# B&R Automation Studio project Cognex_V1_5
Automation Studio 4.6.3.55 SP

## Configuration PP500_15

CPU , AutomationRuntime H4.06, Build 4.1.2, Safety 1.6, Vc V4.05.6

### Task classes (Cpu.sw)
```
Cyclic#8:
  Cognex <- Cognex.prg
  CognexVisN <- CognexVisNativeMode.prg
  CognexVisC <- CognexVisCommissioning.prg
  CognexVisA <- CognexVisArchive.prg
  CognexVisM <- CognexVisMain.prg
VcDataObjects: Visu <- Visu.dob
Binaries: vcclbox, vcctext, vcrt, vcresman, vccbar, vccstr, vccurl, vcchtml, vcpfmtcx, vcptelo, vcfile, vcdsint, vcpdsw, vccshape, arial, vccbmp, vcmgr, vcpdi855, vcshared, Visu01, vcdsloc, vcfntttf, vccovl, vctcal, arialbd, vcalarm, vcpfpp50, vccnum, vccline, vcpdi815, vccbtn, vcgclass, vcbclass, vcxml, Visu02, Visu03, visvc, vcpdvnc, vcnet, arconfig, sysconf, ashwd, asfw, iomap, vccalarm
Libraries: asieccon, asstring, astime, runtime, FileIO, Visapi, standard, BR_ATL_BMP, BR_ATL_LOG, sys_lib, dataobj, BR_ATL_COG, AsTCP, ethernet, AsICMP
```

## Configuration X20CPU1484

CPU , AutomationRuntime V3.08, Build 4.1.2, Vc V3.95.6

### Task classes (Cpu.sw)
```
Cyclic#8 (cycle 4000 us, tolerance 30004000 us):
  Cognex <- Cognex.prg
  CognexVisM <- CognexVisMain.prg
  CognexVisA <- CognexVisArchive.prg
  CognexVisN <- CognexVisNativeMode.prg
VcDataObjects: Visu <- Visu.dob
Binaries: vcdsint, vcclbox, Visu03, vcctext, vcrt, vccnum, vccbar, vccstr, vccurl, vcchtml, vcresman, vcfile, vcpfx20, vcpdsw, vccshape, arial, vccbmp, vcmgr, visvc, Visu01, vcdsloc, vcfntttf, vccovl, vctcal, arialbd, vcalarm, vccline, vcshared, vccbtn, vcgclass, vcbclass, vcxml, vcnet, vcpdvnc, Visu02, ashwd, sysconf, asfw, arconfig, iomap
Libraries: sys_lib, asstring, BR_ATL_LOG, Operator, Runtime, AsTime, AsIecCon, FileIO, Visapi, standard, BR_ATL_BMP, ashw, dataobj, BR_ATL_COG, AsTCP
```

### Hardware
```
In-Sight : FBE.0000031D_In-Sight-7000 v1.0 (OrderNumber=In-Sight)  [PLK1 -> PLC1.IF3 (NodeNumber=1)]
  Supervision = off
  p2000s01_direction = wo
  p2000s02_direction = wo
  p2001s01_direction = ro
  p2001s02_direction = ro
  p2010s01_direction = ro
  p2011s01_direction = ro
  p2011s02_direction = ro
  p2011s03_direction = ro
  p2011s04_direction = ro
  p2011s05_direction = ro
  p2011s06_direction = ro
  p2011s07_direction = ro
  p2011s08_direction = ro
  p2011s09_direction = ro
  p2011s0A_direction = ro
  p2011s0B_direction = ro
  p2021s01_direction = wo
  p2021s02_direction = wo
  p2021s03_direction = wo
  p2030s01_value = 1500
PLC1 : X20CP1486 v1.1.2.0
  Connector IF2:
    ActivateDevice = 1
    Mode = DHCP Server
    InternetAddress = 192.168.0.10
    SubnetMask = 255.255.255.0
    Lease1
    LeaseName1 = Cognex
    LeaseStartAddress1 = 192.168.0.50
    LeaseStopAddress1 = 192.168.0.55
    LeaseSubnetMask1 = 255.255.255.0
    Vnc1
    VncVcObjectName1 = Visu
    VncPortNumber1 = 5900
    VncMaxConnections1 = 1
    VncRefreshRate1 = 500
    VncConnectionTimeout1 = 4
    VncAuthentication1 = 1
    VncPasswordViewOnly1 = r
    VncPasswordViewControl1 = w
  Connector IF3:
    MtuSize = 1500
    CycleTime = 800
    InternetAddress = 192.168.2.1
    SubnetMask = 255.255.255.0
  UserRamSize = 100000
  RemMemSize = 32000
  Connections = 6
  TimerDeviceType = EPLX2X
  TaskClassIdleTime = 800
  Cyclic1Duration = 2400
  Cyclic1Tolerance = 12000
  Cyclic3Duration = 50400
  Cyclic3Tolerance = 50400
  Cyclic8Duration = 4000
  Cyclic8Tolerance = 30004000
  TimerDevice = PLC1.IF3
```

### IoMap.iom - PLC1/IoMap.iom
```iecst
(********************************************************************
 * COPYRIGHT --
 ********************************************************************
 * File: IoMap.iom
 * Author: strickers
 * Created: May 07, 2012
 ********************************************************************
 * IO mapping file
 ********************************************************************)
VAR_CONFIG
	CognexVisM:CameraIsConnected AT %IX."In-Sight".ModuleOk;
	Cognex:tmpBarcodeRead1 AT %ID."In-Sight".InspectionResults_I2011_S01;
	Cognex:tmpBarcodeRead2 AT %ID."In-Sight".InspectionResults_I2011_S02;
	Cognex:tmpBarcodeRead3 AT %ID."In-Sight".InspectionResults_I2011_S03;
	Cognex:tmpBarcodeWrite1 AT %QD."In-Sight".UserData_I2021_S01;
	Cognex:tmpBarcodeWrite2 AT %QD."In-Sight".UserData_I2021_S02;
	Cognex:tmpBarcodeWrite3 AT %QD."In-Sight".UserData_I2021_S03;
	Cognex:cognex1cmd AT %QD."In-Sight".Control_I2000_S01;
	cognex_1.cmd.job_id AT %QW."In-Sight".JobLoadID_I2000_S02;
	Cognex:cognex1sta AT %ID."In-Sight".Status_I2001_S01;
	cognex_1.sta.job_id AT %IW."In-Sight".CurrentJobID_I2001_S02;
	Cognex:tmpTextRead1 AT %ID."In-Sight".InspectionResults_I2011_S04;
	Cognex:tmpTextRead2 AT %ID."In-Sight".InspectionResults_I2011_S05;
	Cognex:tmpTextRead3 AT %ID."In-Sight".InspectionResults_I2011_S06;
	Cognex:tmpData1 AT %ID."In-Sight".InspectionResults_I2011_S07;
	Cognex:tmpData2 AT %ID."In-Sight".InspectionResults_I2011_S08;
	Cognex:tmpData3 AT %ID."In-Sight".InspectionResults_I2011_S09;
	Cognex:tmpData4 AT %ID."In-Sight".InspectionResults_I2011_S0A;
	Cognex:tmpData5 AT %ID."In-Sight".InspectionResults_I2011_S0B;
END_VAR
```

## Logical view

Binary libraries used (declarations not repeated): AsICMP

### Global.typ
```iecst
(********************************************************************
 * COPYRIGHT --
 ********************************************************************
 * File: Global.typ
 * Author: strickers
 * Created: May 02, 2012
 ********************************************************************
 * Global data types of project Cognex_1
 ********************************************************************)

TYPE
	cognex_sta_typ : 	STRUCT
		connected_eth : BOOL;
		connected_plk : BOOL;
		trigger_ready : BOOL;
		trigger_ack : BOOL;
		acquiring : BOOL;
		missed_acq : BOOL;
		offline_reason : USINT;
		online : BOOL;
		inspecting : BOOL;
		inspecting_complete : BOOL;
		results_buffer_overrun : BOOL;
		results_valid : BOOL;
		job_loading : BOOL;
		job_load_complete : BOOL;
		job_load_failed : BOOL;
		set_user_data_ack : BOOL;
		exposure_complete : BOOL;
		soft_event_ack : USINT;
		job_id : UINT;
	END_STRUCT;
	cognex_cmd_typ : 	STRUCT
		trigger_enable : BOOL;
		trigger : BOOL;
		buffer_result_enable : BOOL;
		inspection_result_ack : BOOL;
		init_job_load : BOOL;
		set_offline : BOOL;
		set_user_data : BOOL;
		clr_exposure_complete : BOOL;
		soft_event : USINT;
		job_id : UINT;
		ping_camera : BOOL;
	END_STRUCT;
	cognex_typ : 	STRUCT
		cmd : cognex_cmd_typ;
		sta : cognex_sta_typ;
	END_STRUCT;
END_TYPE
```

### Global.var
```iecst
(*-------------------------------------------------------------------------------------------------------------------------------------------------------------------------------------------------------------------------*)
VAR
	cognex_1 : cognex_typ; (*Cognex main structure*)
	logbook : ARRAY[0..19] OF STRING[80];
END_VAR
(*-------------------------------------------------------------------------------------------------------------------------------------------------------------------------------------------------------------------------*)
VAR CONSTANT
	PictureWidth : UINT := 200; (*Cognex picture width*)
	PictureHeight : UINT := 150; (*Cognex picture height*)
END_VAR
VAR
	CognexPlkNode : STRING[3] := '1'; (*Powerlink node number for Cognex camera*)
	CognexEthIP : STRING[30] := '192.168.0.220'; (*IP address for camera when connected to Ethernet port*)
END_VAR
(*-------------------------------------------------------------------------------------------------------------------------------------------------------------------------------------------------------------------------*)
VAR
	VIS_HIDDEN : UINT := 1; (*Visualization status constants*)
END_VAR
VAR CONSTANT
	VIS_INACTIVE : UINT := 2;
	VIS_ACTIVE : UINT := 0;
END_VAR
(*-------------------------------------------------------------------------------------------------------------------------------------------------------------------------------------------------------------------------*)
VAR CONSTANT
	READ_ID1 : USINT := 1;
	READ_CFG : USINT := 2;
	WRITE_ID1 : USINT := 1;
	WRITE_ID2 : USINT := 2;
	WRITE_ID3 : USINT := 3;
	WRITE_CFG : USINT := 4;
END_VAR
(*-------------------------------------------------------------------------------------------------------------------------------------------------------------------------------------------------------------------------*)
VAR CONSTANT
	NONE : USINT := 0;
	CMD_INFO : USINT := 1;
	CMD_STATUS : USINT := 2;
	CMD_DELETE_JOBID3 : USINT := 3;
	CMD_SET_OFFLINE : USINT := 4;
END_VAR
```

### Program Logical/Cognex

#### Cognex.ab
```automation-basic
(********************************************************************
 * COPYRIGHT --
 ********************************************************************
 * Program: NewProgram
 * File: NewProgram.ab
 * Author: strickers
 * Version: 1.0
 * This task has the following purpose
 * - Transfer text string from sample into PLC variable
 * - Transfer barcode string from sample into PLC variable
 * - Transfer compare string to Cognex variable
 * - Transfer add on data (pass, angle, time) into PLC variables
 * - Transfer camera status into bool structure
 * - Transfer camera commands from PLC structure to camera
 ********************************************************************)

PROGRAM _INIT
		strcpy(ADR(strBarcodeWrite), ADR("ABA122"))
END_PROGRAM

PROGRAM _CYCLIC
	(* -------------------------------------------------------------------- *)
	(* Send ping to camera			 										*)
	IF (cognex_1.cmd.ping_camera) THEN
		ICMPping_0.enable 	= 1
		ICMPping_0.pHost 	= adr(CognexEthIP)
		ICMPping_0.timeout 	= 20
		ICMPping_0 FUB IcmpPing()
		IF(ICMPping_0.status <> 65535) THEN
			cognex_1.cmd.ping_camera = 0
			IF(ICMPping_0.status = 0) THEN
				cognex_1.sta.connected_eth = 1
			ELSE
				cognex_1.sta.connected_eth = 0
			ENDIF
		ENDIF
	ENDIF

	IF(cognex_1.sta.online) THEN
	(* -------------------------------------------------------------------- *)
	(* Transfer text string			 										*)
	memcpy(ADR(strTextRead)+0,ADR(tmpTextRead1), 4)
	memcpy(ADR(strTextRead)+4,ADR(tmpTextRead2), 4)
	memcpy(ADR(strTextRead)+8,ADR(tmpTextRead3), 4)

	(* -------------------------------------------------------------------- *)
	(* Transfer barcode string			 									*)
	memcpy(ADR(strBarcodeRead)+0,ADR(tmpBarcodeRead1), 4)
	memcpy(ADR(strBarcodeRead)+4,ADR(tmpBarcodeRead2), 4)
	memcpy(ADR(strBarcodeRead)+8,ADR(tmpBarcodeRead3), 4)

	memcpy(ADR(tmpBarcodeWrite1), ADR(strBarcodeWrite)+0, 4)
	memcpy(ADR(tmpBarcodeWrite2), ADR(strBarcodeWrite)+4, 4)
	memcpy(ADR(tmpBarcodeWrite3), ADR(strBarcodeWrite)+8, 4)
	IF(strcmp(ADR(strBarcodeWrite), ADR(strBarcodeWriteOld)) <> 0) THEN
		cognex_1.cmd.set_user_data = 1
		strcpy(ADR(strBarcodeWriteOld), ADR(strBarcodeWrite))
	ELSE
		cognex_1.cmd.set_user_data = 0
	ENDIF
	ENDIF

	(* -------------------------------------------------------------------- *)
	(* Transfer additonal data			 									*)
	memcpy(ADR(FixturePass),ADR(tmpData1)+0, 1)
	memcpy(ADR(BarcodePass),ADR(tmpData1)+1, 1)
	memcpy(ADR(TextPass),ADR(tmpData1)+2, 1)
	memcpy(ADR(ComparePass),ADR(tmpData1)+3, 1)
	memcpy(ADR(TextExecutionTime),ADR(tmpData2), 4)
	memcpy(ADR(BarcodeFixtureAngle),ADR(tmpData3), 4)
	memcpy(ADR(JobExecutionTime),ADR(tmpData4), 4)
	memcpy(ADR(JobPass),ADR(tmpData5)+0, 1)

	(* -------------------------------------------------------------------- *)
	(* Copy status data into structure 										*)
	cognex_1.sta.trigger_ready 			= cognex1sta.0
	cognex_1.sta.trigger_ack 			= cognex1sta.1
	cognex_1.sta.acquiring 				= cognex1sta.2
	cognex_1.sta.missed_acq 			= cognex1sta.3
	cognex_1.sta.offline_reason.0 		= cognex1sta.4
	cognex_1.sta.offline_reason.1 		= cognex1sta.5
	cognex_1.sta.offline_reason.2 		= cognex1sta.6
	cognex_1.sta.online 				= cognex1sta.7
	cognex_1.sta.inspecting 			= cognex1sta.8
	cognex_1.sta.inspecting_complete	= cognex1sta.9
	cognex_1.sta.results_buffer_overrun = cognex1sta.10
	cognex_1.sta.results_valid 			= cognex1sta.11
	cognex_1.sta.job_loading 			= cognex1sta.12
	cognex_1.sta.job_load_complete 		= cognex1sta.13
	cognex_1.sta.job_load_failed 		= cognex1sta.14
	cognex_1.sta.set_user_data_ack 		= cognex1sta.16
	cognex_1.sta.exposure_complete 		= cognex1sta.19
	cognex_1.sta.soft_event_ack.0 		= cognex1sta.24
	cognex_1.sta.soft_event_ack.1 		= cognex1sta.25
	cognex_1.sta.soft_event_ack.2 		= cognex1sta.26
	cognex_1.sta.soft_event_ack.3 		= cognex1sta.27
	cognex_1.sta.soft_event_ack.4 		= cognex1sta.28
	cognex_1.sta.soft_event_ack.5 		= cognex1sta.29
	cognex_1.sta.soft_event_ack.6 		= cognex1sta.30
	cognex_1.sta.soft_event_ack.7 		= cognex1sta.31

	(* -------------------------------------------------------------------- *)
	(* Copy command data from structure 									*)
	cognex1cmd.0 = cognex_1.cmd.trigger_enable
	cognex1cmd.1 = cognex_1.cmd.trigger
	cognex1cmd.2 = cognex_1.cmd.buffer_result_enable
	cognex1cmd.3 = cognex_1.cmd.inspection_result_ack
	cognex1cmd.4 = cognex_1.cmd.init_job_load
	cognex1cmd.7 = cognex_1.cmd.set_offline
	cognex1cmd.16 = cognex_1.cmd.set_user_data
	cognex1cmd.19 = cognex_1.cmd.clr_exposure_complete
	cognex1cmd.24 = cognex_1.cmd.soft_event.0
	cognex1cmd.25 = cognex_1.cmd.soft_event.1
	cognex1cmd.26 = cognex_1.cmd.soft_event.2
	cognex1cmd.27 = cognex_1.cmd.soft_event.3
	cognex1cmd.28 = cognex_1.cmd.soft_event.4
	cognex1cmd.29 = cognex_1.cmd.soft_event.5
	cognex1cmd.30 = cognex_1.cmd.soft_event.6
	cognex1cmd.31 = cognex_1.cmd.soft_event.7

	(* -------------------------------------------------------------------- *)
	(* Generate logbook entries for camera events 							*)
	IF(EDGEPOS(cognex_1.sta.trigger_ready)) THEN
		NewLogEntry("Trigger is ready", ADR(logbook), 20)
	ENDIF
	IF(EDGEPOS(cognex_1.sta.inspecting)) THEN
		NewLogEntry("Trigger was acknowledged", ADR(logbook), 20)
	ENDIF
	IF(EDGEPOS(cognex_1.sta.acquiring)) THEN
		NewLogEntry("-----------------------------------------------------", ADR(logbook), 20)
		NewLogEntry("Aquiring new picture", ADR(logbook), 20)
	ENDIF
	IF(EDGEPOS(cognex_1.sta.missed_acq)) THEN
		NewLogEntry("Aquiring new picture missed", ADR(logbook), 20)
	ENDIF
	IF(EDGEPOS(cognex_1.sta.online)) THEN
		NewLogEntry("Camera is online", ADR(logbook), 20)
	ENDIF
	IF(EDGENEG(cognex_1.sta.online)) THEN
		NewLogEntry("Camera is offline", ADR(logbook), 20)
	ENDIF
	IF(EDGEPOS(cognex_1.sta.inspecting)) THEN
		NewLogEntry("Starting inspecting picture", ADR(logbook), 20)
	ENDIF
	IF(cognex_1.sta.inspecting_complete <> tmp_inspecting_complete) THEN
		NewLogEntry("Completed inspecting picture", ADR(logbook), 20)
		tmp_inspecting_complete = cognex_1.sta.inspecting_complete
	ENDIF
	IF(EDGEPOS(cognex_1.sta.results_buffer_overrun)) THEN
		NewLogEntry("Results buffer overrun", ADR(logbook), 20)
	ENDIF
	IF(EDGEPOS(cognex_1.sta.results_valid)) THEN
		NewLogEntry("Results is valid", ADR(logbook), 20)
	ENDIF
	IF(EDGEPOS(cognex_1.sta.job_loading)) THEN
		NewLogEntry("Loading new job", ADR(logbook), 20)
	ENDIF
	IF(cognex_1.sta.job_load_complete <> tmp_job_complete) THEN
		NewLogEntry("Loading new job complete", ADR(logbook), 20)
		tmp_job_complete = cognex_1.sta.job_load_complete
		IF(cognex_1.sta.job_load_failed) THEN
			NewLogEntry("Loading new job failed", ADR(logbook), 20)
		ENDIF
	ENDIF

END_PROGRAM
```

### CognexVisArchive.var
```iecst
(*-------------------------------------------------------------------------------------------------------------------------------------------------------------------------------------------------------------------------*)
VAR
	x : USINT := 0;
	dir_entry_max : USINT := 0;
	dir_data : ARRAY[0..19] OF fiDIR_READ_DATA;
	dir_entry : USINT;
	DirRead_0 : DirRead;
	DirCreate_0 : DirCreate;
	DevLink_0 : DevLink;
END_VAR
(*-------------------------------------------------------------------------------------------------------------------------------------------------------------------------------------------------------------------------*)
VAR
	VChandle : UDINT;
	VCbitmap : REFERENCE TO sVCBitmap;
	VCbitmap_tmp : UDINT;
	VCerror : UINT;
END_VAR
(*-------------------------------------------------------------------------------------------------------------------------------------------------------------------------------------------------------------------------*)
VAR
	step_diag : USINT := 0;
	vkDirRefresh : BOOL := FALSE;
	dir_names : ARRAY[0..19] OF STRING[80];
	dir_name_selected_old : UINT := 0;
	dir_name_selected_max : UINT := 0;
	dir_name_selected : UINT := 0;
END_VAR
(*-------------------------------------------------------------------------------------------------------------------------------------------------------------------------------------------------------------------------*)
VAR CONSTANT
	STP_INIT : USINT := 0;
	STP_DIR_READ : USINT := 3;
	STP_DIR_EVAL : USINT := 4;
	STP_VC_LOAD : USINT := 6;
	STP_VC_SHOW : USINT := 7;
	STP_VC_FREE : USINT := 8;
	STP_ERROR : USINT := 20;
END_VAR
```

### CognexVisMain.var
```iecst
(*-------------------------------------------------------------------------------------------------------------------------------------------------------------------------------------------------------------------------*)
VAR
	vsCameraConnectedPlk : UINT;
	vsCameraOnline : UINT;
	vsCameraChangeJob : UINT;
	vsCameraTrigger : UINT;
	vsCameraJob1 : UINT;
	vsErrorReset : UINT := 1;
	vkErrorReset : BOOL;
END_VAR
(*-------------------------------------------------------------------------------------------------------------------------------------------------------------------------------------------------------------------------*)
VAR
	step_pic : USINT := 0;
	x : USINT := 0;
	DirRead_0 : DirRead;
	DirCreate_0 : DirCreate;
	FileDelete_0 : FileDelete;
	DevLink_0 : DevLink;
	TON_10ms_0 : TON_10ms;
	DTnow : DATE_AND_TIME;
	DTGetTime_0 : DTGetTime;
	DTGetTimeTollerance : UDINT;
	file_converted : STRING[260];
	file_newest : STRING[260];
	dir_wait_time : UDINT := 0; (*Wait timer for camera picture*)
	dir_timeout : UDINT := 5000; (*Picture timeout in ms*)
	dir_cleanup : BOOL; (*Flag for folder clean up*)
	dir_data_oldest : fiDIR_READ_DATA; (*File information for oldest file*)
	dir_data_newest : fiDIR_READ_DATA; (*File information for newest file*)
	dir_entry_max : USINT := 0; (*Max number of files, depends on next array size*)
	dir_data : ARRAY[0..19] OF fiDIR_READ_DATA;
	dir_entry : USINT;
END_VAR
(*-------------------------------------------------------------------------------------------------------------------------------------------------------------------------------------------------------------------------*)
VAR
	VChandle : UDINT;
	VCbitmap : REFERENCE TO sVCBitmap;
	VCbitmap_tmp : UDINT;
	VCerror : UINT;
	BmpConvert_0 : BmpConvert;
END_VAR
(*-------------------------------------------------------------------------------------------------------------------------------------------------------------------------------------------------------------------------*)
VAR CONSTANT
	STP_INIT : USINT := 0;
	STP_RESULT : USINT := 1;
	STP_WAIT : USINT := 2;
	STP_DIR_READ : USINT := 3;
	STP_DIR_EVAL : USINT := 4;
	STP_VC_CONVERT : USINT := 5;
	STP_VC_LOAD : USINT := 6;
	STP_VC_SHOW : USINT := 7;
	STP_VC_FREE : USINT := 8;
	STP_BMP_DELETE : USINT := 9;
	STP_BMP_CLEANUP : USINT := 10;
	STP_ERROR : USINT := 20;
END_VAR
```

### Program Logical/CognexVisNativeMode

#### CognexVisNativeMode.ab
```automation-basic
(********************************************************************
 * COPYRIGHT --
 ********************************************************************
 * Author: strickers
 * Version: 1.0
 * This task has the following purpose
 * - Connect to Cognex telnet (Native interface)
 * - Read command_status information
 * - Read and write camera jobs
 * - Read and write camera settings
 ********************************************************************)

PROGRAM _INIT
	(* --------------------------------------------------------------------------------------------------------- *)
	(* Create file device for Cognex files and configuration files *)
	LOOP
		DevLink_0.enable 	= 1
		DevLink_0.pDevice 	= ADR("root")
		DevLink_0.pParam 	= ADR("/DEVICE=C:\\")
		DevLink_0 FUB DevLink()
		EXITIF(DevLink_0.status <> 65535)
	ENDLOOP
	(* --------------------------------------------------------------------------------------------------------- *)
	(* Create folder for Cognex files and configuration files *)
	LOOP
		DirCreate_0.enable 	= 1
		DirCreate_0.pDevice = ADR("root")
		DirCreate_0.pName 	= ADR("cognex_files")
		DirCreate_0 FUB DirCreate()
		EXITIF(DirCreate_0.status <> 65535)
	ENDLOOP
	(* --------------------------------------------------------------------------------------------------------- *)
	(* Create file device for Cognex files and configuration files *)
	LOOP
		DevLink_0.enable 	= 1
		DevLink_0.pDevice 	= ADR("CognexFiles")
		DevLink_0.pParam 	= ADR("/DEVICE=C:\\cognex_files")
		DevLink_0 FUB DevLink()
		EXITIF(DevLink_0.status <> 65535)
	ENDLOOP
	NativeModeStatus = VIS_INACTIVE
	TransferProgressStatus = VIS_HIDDEN
	strcat(ADR(CognexPlkIP), ADR(CognexPlkNode))
END_PROGRAM

PROGRAM _CYCLIC

(* --------------------------------------------------------------------------------------------------------- *)
(* Connect to camera
(* --------------------------------------------------------------------------------------------------------- *)
IF(EDGEPOS(vkNativeModeConnect)) THEN
	NewLogEntry("Connecting to camera...", ADR(logbook), 20)
ENDIF
IF(EDGENEG(cognex_1.sta.connected_plk) AND (NativeModeLoggedIn = TRUE)) THEN
	vkNativeModeConnect = TRUE
ENDIF
IF(vkNativeModeConnect = TRUE) THEN
	IF(NativeModeLoggedIn = FALSE) THEN
		NativeModeLogin_0.enable = 1
		NativeModeLogin_0.ip = ADR(CognexPlkIP)
		NativeModeLogin_0 FUB NativeModeLogin()
		IF(NativeModeLogin_0.status <> 65535) THEN
			IF(NativeModeLogin_0.status = 0) THEN
				NewLogEntry("Loggged into camera", ADR(logbook), 20)
				NativeModeLoggedIn	= TRUE
				NativeModeStatus 	= VIS_ACTIVE
			ELSE
				NewLogEntry("Failed to log into camera", ADR(logbook), 20)
				vsErrorReset = VIS_ACTIVE
			ENDIF
			vkNativeModeConnect = FALSE
		endif
	ELSE
(* --------------------------------------------------------------------------------------------------------- *)
(* Disconnect from camera
(* --------------------------------------------------------------------------------------------------------- *)
		NativeModeLogout_0.enable = 1
		NativeModeLogout_0.ident = NativeModeLogin_0.ident
		NativeModeLogout_0 FUB NativeModeLogout()
		IF(NativeModeLogout_0.status <> 65535) THEN
			NewLogEntry("Loggged out of camera", ADR(logbook), 20)
			NativeModeReadFile_0.enable = 0
			NativeModeReadFile_0 FUB NativeModeReadFile()
			NativeModeWriteFile_0.enable = 0
			NativeModeWriteFile_0 FUB NativeModeWriteFile()

			vsTransferProgress 		= 0
			TransferProgressStatus  = VIS_HIDDEN
			vkTransferWrite 		= NONE
			vkTransferRead 			= NONE
			vkTransferCancel 		= FALSE

			NativeModeLogin_0.enable = 0
			NativeModeLogin_0 FUB NativeModeLogin()
			NativeModeStatus 	= VIS_INACTIVE
			NativeModeLoggedIn	= FALSE
			vkNativeModeConnect	= FALSE
		ENDIF
	ENDIF
ENDIF

(* --------------------------------------------------------------------------------------------------------- *)
(* Use command interface for Cognex camera
(* --------------------------------------------------------------------------------------------------------- *)
IF(NaticeModeCommand = CMD_INFO) THEN
	NativeModeCommand_0.command = ADR("GI")
ENDIF
IF(NaticeModeCommand = CMD_STATUS) THEN
	NativeModeCommand_0.command 	= ADR("EV GetMSBuffer(0)")
ENDIF
IF(NaticeModeCommand = CMD_DELETE_JOBID3) THEN
	NativeModeCommand_0.command 	= ADR("DJ3")
ENDIF
IF(NaticeModeCommand <> NONE) THEN
	NativeModeCommand_0.enable 		= 1
	NativeModeCommand_0.ident 		= NativeModeLogin_0.ident
	NativeModeCommand_0.out_data 	= ADR(data)
	NativeModeCommand_0.out_size 	= SIZEOF(data)
	NativeModeCommand_0 FUB NativeModeCommand()
	NativeModeStatus = VIS_INACTIVE
	IF(NativeModeCommand_0.status <> 65535) THEN
		IF(NativeModeCommand_0.status = 0) THEN
			NewLogEntry("Command finished", ADR(logbook), 20)
			(* Separate data stream by \r\n and split into strings *)
			NativeModeCommandStatus = NativeModeSeparateData(ADR(data), NativeModeCommand_0.in_size, ADR(data_string), SIZEOF(data_string[0]), SIZEOF(data_string)/SIZEOF(data_string[0]))
			(* Check camera responds (1 = The command was executed successfully. 0=Unrecognized command. -2=The command could not be executed. *)
 			IF(NativeModeCommandStatus = 1) THEN
				NativeModeStatus = VIS_ACTIVE
			ELSE
				NewLogEntry("Camera responded with error", ADR(logbook), 20)
				vsErrorReset = VIS_ACTIVE
			ENDIF
		ELSE
			NewLogEntry("Command failed", ADR(logbook), 20)
			vsErrorReset = VIS_ACTIVE
		ENDIF
		NaticeModeCommand = NONE
	ENDIF
ENDIF

(* --------------------------------------------------------------------------------------------------------- *)
(* Read file from Cognex camera
(* --------------------------------------------------------------------------------------------------------- *)
IF EDGEPOS(vkTransferRead = READ_CFG) THEN
	NativeModeReadFile_0.command 	= ADR("RS")
	NativeModeReadFile_0.file_name 	= ADR("settings.dat")
	NewLogEntry("Read job file ID1", ADR(logbook), 20)
ENDIF
IF EDGEPOS(vkTransferRead = READ_ID1) THEN
	NativeModeReadFile_0.command 	= ADR("RJ1")
	NativeModeReadFile_0.file_name 	= ADR("JobFileID1.job")
	NewLogEntry("Read job file ID1", ADR(logbook), 20)
ENDIF
IF(vkTransferRead <> NONE) THEN
	NativeModeReadFile_0.enable 	= 1
	NativeModeReadFile_0.ident 		= NativeModeLogin_0.ident
	NativeModeReadFile_0.device 	= ADR("CognexFiles")
	NativeModeReadFile_0 FUB NativeModeReadFile()
	vsTransferProgress 		= NativeModeReadFile_0.progress
	TransferProgressStatus  = VIS_ACTIVE
	NativeModeStatus 		= VIS_INACTIVE
	IF(NativeModeReadFile_0.status <> 65535) THEN
		IF(NativeModeReadFile_0.status = 0) THEN
			NewLogEntry("Load file finished", ADR(logbook), 20)
			NativeModeStatus = VIS_ACTIVE
		ELSE
			NewLogEntry("Load file failed", ADR(logbook), 20)
			vsErrorReset = VIS_ACTIVE
		ENDIF
		TransferProgressStatus  = VIS_HIDDEN
		vkTransferRead = NONE
	ENDIF
ENDIF

(* --------------------------------------------------------------------------------------------------------- *)
(* Write file to Cognex camera
(* --------------------------------------------------------------------------------------------------------- *)
IF EDGEPOS(vkTransferWrite = WRITE_ID3) THEN
	NativeModeWriteFile_0.command 	= ADR("WJ3")
	NativeModeWriteFile_0.file_name = ADR("3_Powerlink.job")
	NewLogEntry("Write job file ID3", ADR(logbook), 20)
ENDIF
IF(vkTransferWrite <> NONE) THEN
	NativeModeWriteFile_0.enable 	= 1
	NativeModeWriteFile_0.ident 	= NativeModeLogin_0.ident
	NativeModeWriteFile_0.device 	= ADR("CognexFiles")
	NativeModeWriteFile_0 FUB NativeModeWriteFile()
	TransferProgressStatus  = VIS_ACTIVE
	vsTransferProgress 		= NativeModeWriteFile_0.progress
	NativeModeStatus 		= VIS_INACTIVE
	IF(NativeModeWriteFile_0.status <> 65535) THEN
		IF(NativeModeWriteFile_0.status = 0) THEN
			NewLogEntry("Write file finished", ADR(logbook), 20)
			NativeModeStatus = VIS_ACTIVE
		ELSE
			NewLogEntry("Write file failed", ADR(logbook), 20)
			vsErrorReset = VIS_ACTIVE
		ENDIF
		TransferProgressStatus  = VIS_HIDDEN
		vkTransferWrite = NONE
	ENDIF
ENDIF

(* --------------------------------------------------------------------------------------------------------- *)
(* Error handling and reset
(* --------------------------------------------------------------------------------------------------------- *)
IF (vkErrorReset) THEN
	IF(NativeModeLogin_0.status <> 0) THEN
		NativeModeLoggedIn	= TRUE
		vkNativeModeConnect = TRUE
	ENDIF
	vsTransferProgress = 0
	NativeModeCommand_0.enable = 0
	NativeModeCommand_0 FUB NativeModeCommand()
	NativeModeReadFile_0.enable = 0
	NativeModeReadFile_0 FUB NativeModeReadFile()
	NativeModeWriteFile_0.enable = 0
	NativeModeWriteFile_0 FUB NativeModeWriteFile()
	memset(ADR(logbook), 0, SIZEOF(logbook))
	NativeModeStatus 	= VIS_ACTIVE
	vsErrorReset 		= VIS_HIDDEN
	vkErrorReset 		= 0
ENDIF

END_PROGRAM
```

### Library Logical/Libraries/BR_ATL_COG (ANSIC, version 1.10.0)
Depends on: AsTCP, standard, FileIO

#### BR_ATL_COG.typ - Exported data types
```iecst
(********************************************************************
 * COPYRIGHT --
 ********************************************************************
 * Library: BR_ATL_COG
 * File: BR_ATL_COG.typ
 * Author: strickers
 * Created: July 16, 2012
 ********************************************************************
 * Data types of library BR_ATL_COG
 ********************************************************************)

TYPE
	typ_cog_login_internal : 	STRUCT
		TELclose : TcpClose;
		TELopen : TcpOpen;
		TELconnect : TcpClient;
		TELwrite : TcpSend;
		TELread : TcpRecv;
		tmpSTR1 : STRING[40];
		tmpSTR2 : STRING[40];
		step_forward : USINT;
		step : USINT;
		TON_10ms_0 : TON_10ms;
		out_size : UINT;
		tmpSTR : STRING[400];
		err_step : USINT;
	END_STRUCT;
	typ_cog_logout_internal : 	STRUCT
		edge_enable : BOOL;
		TELclose : TcpClose;
	END_STRUCT;
	typ_cog_load_file_internal : 	STRUCT
		step : USINT;
		TcpRecv_0 : TcpRecv;
		TcpSend_0 : TcpSend;
		FileClose_0 : FileClose;
		FileWrite_0 : FileWrite;
		FileCreate_0 : FileCreate;
		FileDelete_0 : FileDelete;
		TON_10ms_0 : TON_10ms;
		err_step : USINT;
		command : STRING[100];
		add_byte : USINT;
		file_offset : UDINT;
		data_CRC : UINT;
		data_header : UDINT;
		data_size : UDINT;
		data_read_odd : BOOL;
		data_curr : UDINT;
		data_received : UDINT;
		file_CRC : UINT;
		file_size : UDINT;
		file_name : STRING[80];
		is_header : BOOL;
		command_status : INT;
	END_STRUCT;
	typ_cog_write_file_internal : 	STRUCT
		step : USINT;
		TcpRecv_0 : TcpRecv;
		TcpSend_0 : TcpSend;
		FileClose_0 : FileClose;
		FileRead_0 : FileRead;
		FileOpen_0 : FileOpen;
		FileWrite_0 : FileWrite;
		FileCreate_0 : FileCreate;
		FileDelete_0 : FileDelete;
		TON_10ms_0 : TON_10ms;
		err_step : USINT;
		add_byte : USINT;
		file_offset1 : UDINT;
		test : STRING[200];
		file_offset : UDINT;
		data_CRC : UINT;
		data_header : UDINT;
		data_size : UDINT;
		data_read_odd : BOOL;
		data_curr : UDINT;
		data_send_offset : USINT;
		data_received : UDINT;
		file_CRC : UINT;
		file_size : UDINT;
		file_name : STRING[80];
		firstrun : BOOL;
		lastrun : BOOL;
		command_status : INT;
	END_STRUCT;
	typ_cog_cmd_internal : 	STRUCT
		step : USINT;
		TcpRecv_0 : TcpRecv;
		TcpSend_0 : TcpSend;
		command : STRING[100];
		TON_10ms_0 : TON_10ms;
		err_step : USINT;
	END_STRUCT;
END_TYPE
```

#### BR_ATL_COG.fun - Exported functions and function blocks
```iecst
(********************************************************************
 * COPYRIGHT --
 ********************************************************************
 * Library: BR_ATL_COG
 * File: BR_ATL_COG.fun
 * Author: strickers
 * Created: July 16, 2012
 ********************************************************************
 * Functions and function blocks of library BR_ATL_COG
 ********************************************************************)

FUNCTION NativeModeCRC : UINT
	VAR_INPUT
		cword : UINT;
		buffer : UDINT;
		size : UDINT;
	END_VAR
END_FUNCTION

FUNCTION NativeModeSeparateData : INT
	VAR_INPUT
		in_data : UDINT;
		in_size : UDINT;
		out_string : UDINT;
		out_len : UINT;
		out_size : UINT;
	END_VAR
END_FUNCTION

FUNCTION_BLOCK NativeModeWriteFile
	VAR_INPUT
		enable : BOOL;
		ident : UINT;
		command : UDINT;
		file_name : UDINT;
		device : UDINT;
	END_VAR
	VAR_OUTPUT
		progress : USINT;
		status : UINT;
	END_VAR
	VAR
		internal : typ_cog_write_file_internal;
	END_VAR
END_FUNCTION_BLOCK

FUNCTION_BLOCK NativeModeReadFile
	VAR_INPUT
		enable : BOOL;
		ident : UINT;
		command : UDINT;
		file_name : UDINT;
		device : UDINT;
	END_VAR
	VAR_OUTPUT
		progress : USINT;
		status : UINT;
	END_VAR
	VAR
		internal : typ_cog_load_file_internal;
	END_VAR
END_FUNCTION_BLOCK

FUNCTION_BLOCK NativeModeCommand
	VAR_INPUT
		enable : BOOL;
		ident : UINT;
		command : UDINT;
		out_data : UDINT;
		out_size : UINT;
	END_VAR
	VAR_OUTPUT
		in_size : UINT;
		status : UINT;
	END_VAR
	VAR
		internal : typ_cog_cmd_internal;
	END_VAR
END_FUNCTION_BLOCK

FUNCTION_BLOCK NativeModeLogin
	VAR_INPUT
		enable : BOOL;
		ip : UDINT;
	END_VAR
	VAR_OUTPUT
		ident : UINT;
		status : UINT;
	END_VAR
	VAR
		internal : typ_cog_login_internal;
	END_VAR
END_FUNCTION_BLOCK

FUNCTION_BLOCK NativeModeLogout
	VAR_INPUT
		enable : BOOL;
		ident : UINT;
	END_VAR
	VAR_OUTPUT
		status : UINT;
	END_VAR
	VAR
		internal : typ_cog_logout_internal;
	END_VAR
END_FUNCTION_BLOCK
```

#### BR_ATL_COG_LOC.h
```c
/********************************************************************
 * COPYRIGHT --
 ********************************************************************
 * Library: BR_ATL_BMP
 * File: BR_ATL_loc.h
 * Author: strickers
 * Created: May 23, 2012
 *******************************************************************/

#include <bur/plctypes.h>
#include <AsString.h>
#include <string.h>
#include <sys_lib.h>
#include <fileio.h>
#include <astcp.h>
#include <standard.h>

/************************************************************************************************/
/*	Constants definition																		*/
/************************************************************************************************/
/* Constants for main step																		*/
#define STP_INIT			0
#define STP_TEL_OPEN		10
#define STP_TEL_CONNECT		20
#define STP_TEL_READ		30
#define STP_TEL_WRITE		40
#define STP_STATE_LOGIN1	51
#define STP_STATE_LOGIN2	52
#define STP_STATE_LOGIN3	53
#define STP_STATE_LOGIN4	54
#define STP_STATE_LOGIN5	55
#define STP_TCP_SEND		60
#define STP_TCP_RECV		70
#define STP_FILE_OPEN		80
#define STP_FILE_DEL		81
#define STP_FILE_WRITE		82
#define STP_FILE_READ		83
#define STP_FILE_CREATE		84
#define STP_FILE_CLOSE		85
#define STP_ERROR			100

#define CTRL_SEND			1
#define CTRL_ACK			2
#define CTRL_FINISH			3

#define BUSY				65535		/* Constant for status BUSY								*/
#define NO_ENABLE			65534
#define OK					0			/* Constant for status OK								*/
#define TRUE				1
#define FALSE				0

#define ERR_NO_IP_NUM			10000		/* No IP address specified				*/
#define ERR_NO_IDENT			10001		/* No ident specified, attach ident from NativeModeLogin.ident */
#define ERR_NO_CMD				10002		/* Command string is not specified */
#define ERR_DUPLICATE_CMD		10003		/* Multiple commands called at the same time */
#define ERR_SIZE_CMD			10004		/* Command exceeds maximum size of 100 bytes */
#define ERR_RESP_TIMEOUT		10010		/* Cognex camera did not respond to request */
#define ERR_RESP_UNEXPECTED		10011		/* Respond is not expected format */
#define ERR_RESP_HEADER			10012		/* Response header is too small */
#define ERR_RESP_DATA			10020		/* Respond does not contain status */
#define ERR_CAM_CMD_UNKNOWN		10030		/* Unrecognized command */
#define ERR_CAM_NAME_MISS		10031		/* The job filename is missing */
#define ERR_CAM_NAME_UNKNOWN	10032		/* There is no job saved with the given name */
#define ERR_CAM_ACCESS			10033		/* User does not have Full Access to execute the command */
#define ERR_CAM_GENERAL			10039		/* General error message from camera */
#define ERR_FILE_SIZE			10040		/* File exceeds  expected file size */
#define ERR_FILE_CRC			10041		/* The file CRC does not match the data transmitted */

#define MAX_BUFFER_SIZE			1000
#define RESP_TIMEOUT			3000

USINT 	in_buffer[MAX_BUFFER_SIZE];
USINT 	out_buffer[MAX_BUFFER_SIZE];
USINT 	file_buffer[3*MAX_BUFFER_SIZE];
STRING 	data_string[5][50];

static BOOL command_token;					/* Make sure only one command is execute at at time */

unsigned short TranslateCameraError(INT camera_status);
unsigned short NativeModeHexToBin(UDINT in_data, UDINT in_size, UDINT out_data);
unsigned short NativeModeBinToHex(UDINT in_data, UDINT in_size, UDINT out_data, BOOL firstrun);
unsigned short NativeModeCRC(UINT cword, UDINT buffer, UDINT size);

/************************************************************************************************/
/*	Version																						*/
/************************************************************************************************/
/* 1.0 First release																			*/
```

- Library Logical/Libraries/BR_ATL_LOG (ANSIC) (no source held here)

Listed in the project but not available here: Logical/Libraries/BR_ATL_COG/BR_ATL_COG.c, Logical/Libraries/BR_ATL_LOG/BR_ATL_LOG.typ, Logical/Libraries/BR_ATL_LOG/BR_ATL_LOG.var, Logical/Libraries/BR_ATL_LOG/BR_ATL_LOG.fun, Logical/Libraries/BR_ATL_LOG/BR_ATL_LOG.c
